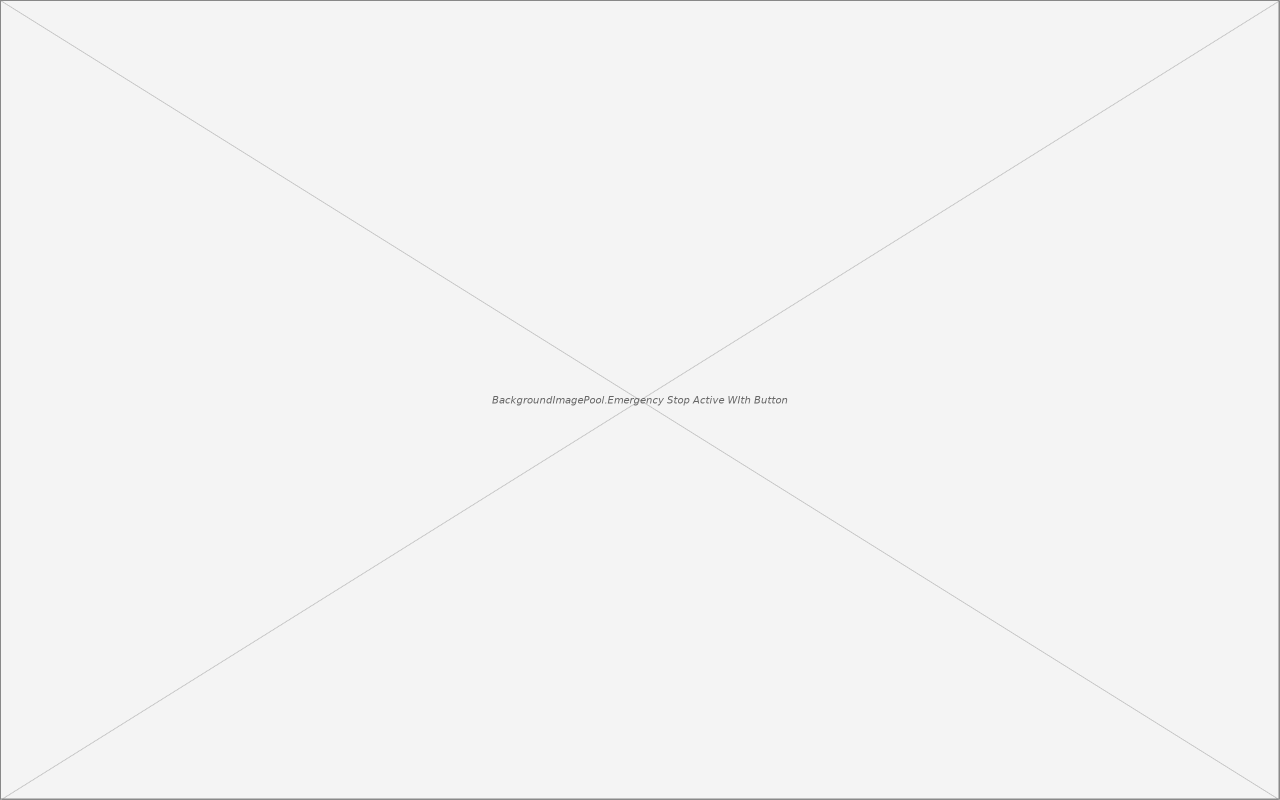
VISUALIZATION BaseScreen  // 1280x800
VAR_IN_OUT
	fbHMIControl : FB_HMIControl ; // hmi control function
END_VAR
    Frame (0,0 1280x800)
        shows BackgroundWithBorder(bCmdSettings := fbHMIControl.bCmdSettings, bHideEstop := fbHMIControl.bHideEStop, bDisableSettings := fbHMIControl.bDisableSettings, bHideBorder := fbHMIControl.bHideBorders)
    Frame (0,0 1280x800), frame switch variable: fbHMIControl.eShownScreen
        shows Idle()
        shows Settings(bCmdParameter := fbHMIControl.bCmdParemeter, nUnitsProduced := System_Library.GVL_Main.nTotalUnitsProduced)
        shows ParameterScreen(bCmdParameter := fbHMIControl.bCmdParemeter)
        shows Manual(bCmdParameter := fbHMIControl.bCmdParemeter)
        shows SemiAuto()
        shows Automatic()
    Image (0,0 1280x800), invisible if: bHideEstop, input disabled if: bHideEstop, image: BackgroundImagePool.Emergency Stop Active WIth Button
END_VISUALIZATION

(* stored: Version 1.1.0.1, ProductVersion 3.1.4024.5
   Visu BaseScreen: Id {4947af5d-5d50-4f16-ab4a-243dcb1607d8} *)
